# EPICS substitutions: bpm_data_combiner_app/Db/bpm.substitutions
file "db/bpm_rec.db"
{
    pattern { VIEW  }
            { out:100ms }
}

file "db/bpm_book_keeping_rec.db"
{
    pattern { VIEW  }
            { out:100ms   }
}

file "db/bpm_with_stats_rec.db"
{
    pattern { VIEW  }
            { out:2s:x }
            { out:2s:y }
}

file "db/bpm_book_keeping_rec.db"
{
    pattern { VIEW  }
            { out:2s }
}
